{attribute 'call_after_init'}
FUNCTION_BLOCK AdsMessageQueue_backup
VAR
	elements : FB_BA_DynamicArray := (uiEntrySize := SIZEOF(POINTER TO AdsMessage), uiMinExpCount := 4); 
	length : INT := 0;
	
	entrySize : UDINT;
END_VAR
(*
this container stores dynamically generated AdsData Structs
AdsData to be added are passed by reference, then this function block allocates a structure to be stored
AdsData are get() by reference and poll() by value
*)

METHOD clear : BOOL
VAR
	i : INT;
	temp : REFERENCE TO AdsMessage;
	tempAdr : POINTER TO AdsMessage;
END_VAR
FOR i:=0 TO length-1 BY 1 DO
	temp := get(index := i, getSize => );
	tempAdr := ADR(temp);
	__DELETE(tempAdr);
END_FOR

elements.Reset();
length := 0;
END_METHOD

METHOD contains : BOOL //check contents, not pointer value
VAR_INPUT
	value : REFERENCE TO AdsMessage;
END_VAR
VAR_OUTPUT
	atIndex : INT;
END_VAR
VAR
	temp : REFERENCE TO AdsMessage;
	i : INT;
END_VAR
IF length = 0 THEN
	contains := FALSE;
	RETURN;
END_IF

FOR i:=0 TO length-1 BY 1 DO
	temp := get(index := i, getSize => );
	
	IF 
		SIZEOF(value) = entrySize AND //same size
		MEMCMP(ADR(temp), ADR(value), SIZEOF(entrySize)) = 0 //same data
	THEN
		contains := TRUE;
		atIndex := i;
		RETURN;
	END_IF
	
END_FOR
contains := FALSE;
END_METHOD

METHOD get : REFERENCE TO AdsMessage
VAR_INPUT
	index : INT;
END_VAR
VAR_OUTPUT
	getSize : UDINT;
END_VAR
IF length = 0 OR index < 0 OR index >= length THEN
	getSize := 0;
ELSE
	elements.GetEntry(diIndex := index, pResultEntry := ADR(get));
	getSize := SIZEOF(get);
END_IF
END_METHOD

METHOD isEmpty : BOOL
VAR_INPUT
END_VAR
isEmpty := length = 0;
END_METHOD

METHOD poll : AdsMessage
VAR_OUTPUT
	getSize : UDINT;
END_VAR
IF length > 0 THEN
	poll := get(index := 0, getSize => getSize);
	elements.RemoveEntry(diIndex := 0);
	
	length := length - 1;
END_IF
END_METHOD

METHOD push : BOOL
VAR_INPUT
	value : REFERENCE TO AdsMessage;
END_VAR
VAR
	temp : POINTER TO AdsMessage;
END_VAR
temp := __NEW(AdsMessage);
temp^ := value;

elements.AddEntryPtr(pEntry := temp);

length := length + 1;
END_METHOD

METHOD set : BOOL
VAR_INPUT
	i : INT;
	value : REFERENCE TO AdsMessage;
END_VAR
VAR
	temp : REFERENCE TO AdsMessage;
END_VAR
IF length = 0 THEN
	RETURN;
END_IF

IF i >= 0 AND i < length THEN
	temp REF= get(i);
	temp := value;
	
	set := TRUE;
END_IF
END_METHOD

{attribute 'call_after_init'}
METHOD setup : BOOL
VAR_INPUT
END_VAR
entrySize := SIZEOF(AdsMessage);
END_METHOD

METHOD size : INT
size := length;
END_METHOD

END_FUNCTION_BLOCK

(* stored: Version 1.1.0.1, ProductVersion 3.1.4024.11
   POU AdsMessageQueue_backup: Id {a2c6cc34-f088-4030-8b1a-a4639cebba3a}, SpecialFunc None
   Method clear: Id {1de2cd01-c8d0-41fb-9b35-16e11b99f099}
   Method contains: Id {800c83e4-5bda-4848-9968-c50585aa1645}
   Method get: Id {c8c2fdb8-2e30-4bba-b479-306ee31032b3}
   Method isEmpty: Id {aee39392-cee2-4fcb-b82e-7998c3f7985d}
   Method poll: Id {f7e4dd30-3002-4a63-84ee-57e3c0aadaf1}
   Method push: Id {818a340a-4145-4bdb-a6ed-d4741d3f0703}
   Method set: Id {71db1b36-34c7-4360-95fd-223b7bda1ee4}
   Method setup: Id {13b14e98-ce4c-4af1-ba64-e90360459dbb}
   Method size: Id {db21a606-0435-46af-a8e7-95ac6d9db747} *)
